SYSTEM DASDAass2_testi (* System Configuration *)
  (* Standard: 61499-1 *)
  (* Version 0.4, 2009-03-05, JHC, Holobloc Inc., Deleted Application. *)
  (* Version 0.3, 2003-12-05, JHC, Rockwell Automation, Renamed from NEWSYSTEM. *)
  (* Version 0.2, 2002-11-05, JHC, Rockwell Automation, Fixed missing (empty) FBD in Application. *)
  (* Version 0.1, 2002-01-17, JHC, Rockwell Automation, Minor cleanup *)
  (* Version 0.0, 2000-05-27, JHC, Rockwell Automation *)
  DEVICE HMI_LAYER : FRAME_DEVICE(BOUNDS := [0,0,200,200])
    RESOURCE HMI_1 : PANEL_RESOURCE(COLS := 1, ROWS := 0)
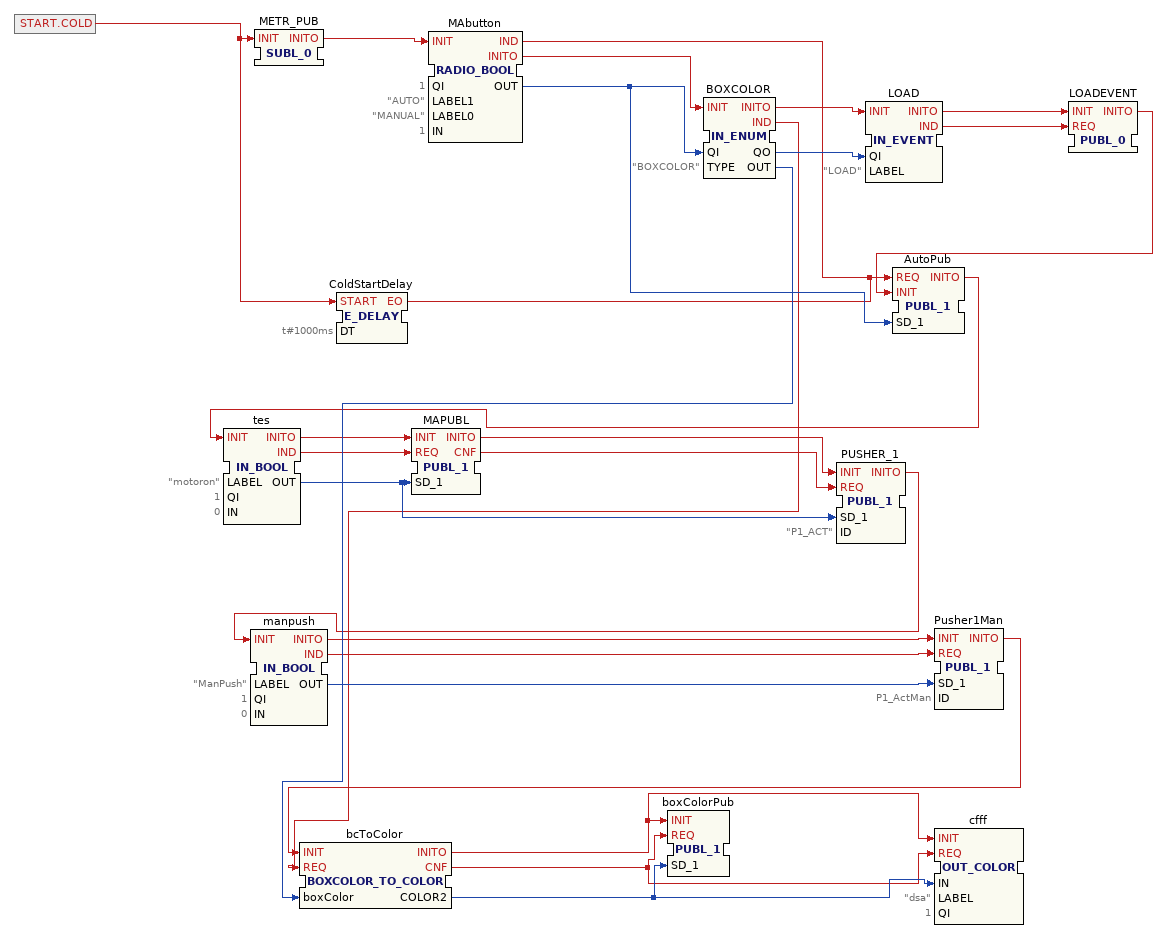
      FBS
        MAbutton : RADIO_BOOL(QI := 1, LABEL1 := "AUTO", LABEL0 := "MANUAL", IN := 1);
        LOAD : IN_EVENT(LABEL := "LOAD");
        LOADEVENT : PUBL_0;
        MAPUBL : PUBL_1;
        tes : IN_BOOL(LABEL := "motoron", QI := 1, IN := 0);
        METR_PUB : SUBL_0;
        PUSHER_1 : PUBL_1(ID := "P1_ACT");
        AutoPub : PUBL_1;
        ColdStartDelay : E_DELAY(DT := t#1000ms);
        manpush : IN_BOOL(LABEL := "ManPush", QI := 1, IN := 0);
        Pusher1Man : PUBL_1(ID := P1_ActMan);
        BOXCOLOR : IN_ENUM(TYPE := "BOXCOLOR");
        bcToColor : BOXCOLOR_TO_COLOR;
        cfff : OUT_COLOR(LABEL := "dsa", QI := 1);
        boxColorPub : PUBL_1;
      END_FBS
      EVENT_CONNECTIONS
        LOAD.INITO TO LOADEVENT.INIT;
        LOAD.IND TO LOADEVENT.REQ;
        START.COLD TO METR_PUB.INIT;
        METR_PUB.INITO TO MAbutton.INIT;
        tes.INITO TO MAPUBL.INIT;
        tes.IND TO MAPUBL.REQ;
        MAPUBL.INITO TO PUSHER_1.INIT;
        MAPUBL.CNF TO PUSHER_1.REQ;
        START.COLD TO ColdStartDelay.START;
        ColdStartDelay.EO TO AutoPub.REQ;
        MAbutton.IND TO AutoPub.REQ;
        LOADEVENT.INITO TO AutoPub.INIT;
        AutoPub.INITO TO tes.INIT;
        PUSHER_1.INITO TO manpush.INIT;
        manpush.INITO TO Pusher1Man.INIT;
        manpush.IND TO Pusher1Man.REQ;
        MAbutton.INITO TO BOXCOLOR.INIT;
        BOXCOLOR.INITO TO LOAD.INIT;
        Pusher1Man.INITO TO bcToColor.INIT;
        bcToColor.INITO TO cfff.INIT;
        bcToColor.CNF TO cfff.REQ;
        BOXCOLOR.IND TO bcToColor.REQ;
        bcToColor.INITO TO boxColorPub.INIT;
        bcToColor.CNF TO boxColorPub.REQ;
      END_CONNECTIONS
      DATA_CONNECTIONS
        tes.OUT TO MAPUBL.SD_1;
        tes.OUT TO PUSHER_1.SD_1;
        MAbutton.OUT TO AutoPub.SD_1;
        manpush.OUT TO Pusher1Man.SD_1;
        MAbutton.OUT TO BOXCOLOR.QI;
        BOXCOLOR.QO TO LOAD.QI;
        bcToColor.COLOR2 TO cfff.IN;
        BOXCOLOR.OUT TO bcToColor.boxColor;
        bcToColor.COLOR2 TO boxColorPub.SD_1;
      END_CONNECTIONS
    END_RESOURCE
  END_DEVICE
  DEVICE VIEW_LAYER : FRAME_DEVICE(BOUNDS := [250,0,900,900])
    RESOURCE VIEW_RES : VIEW_PANEL(DIA := 85, SIZE := [10,8], VERTICAL := 0)
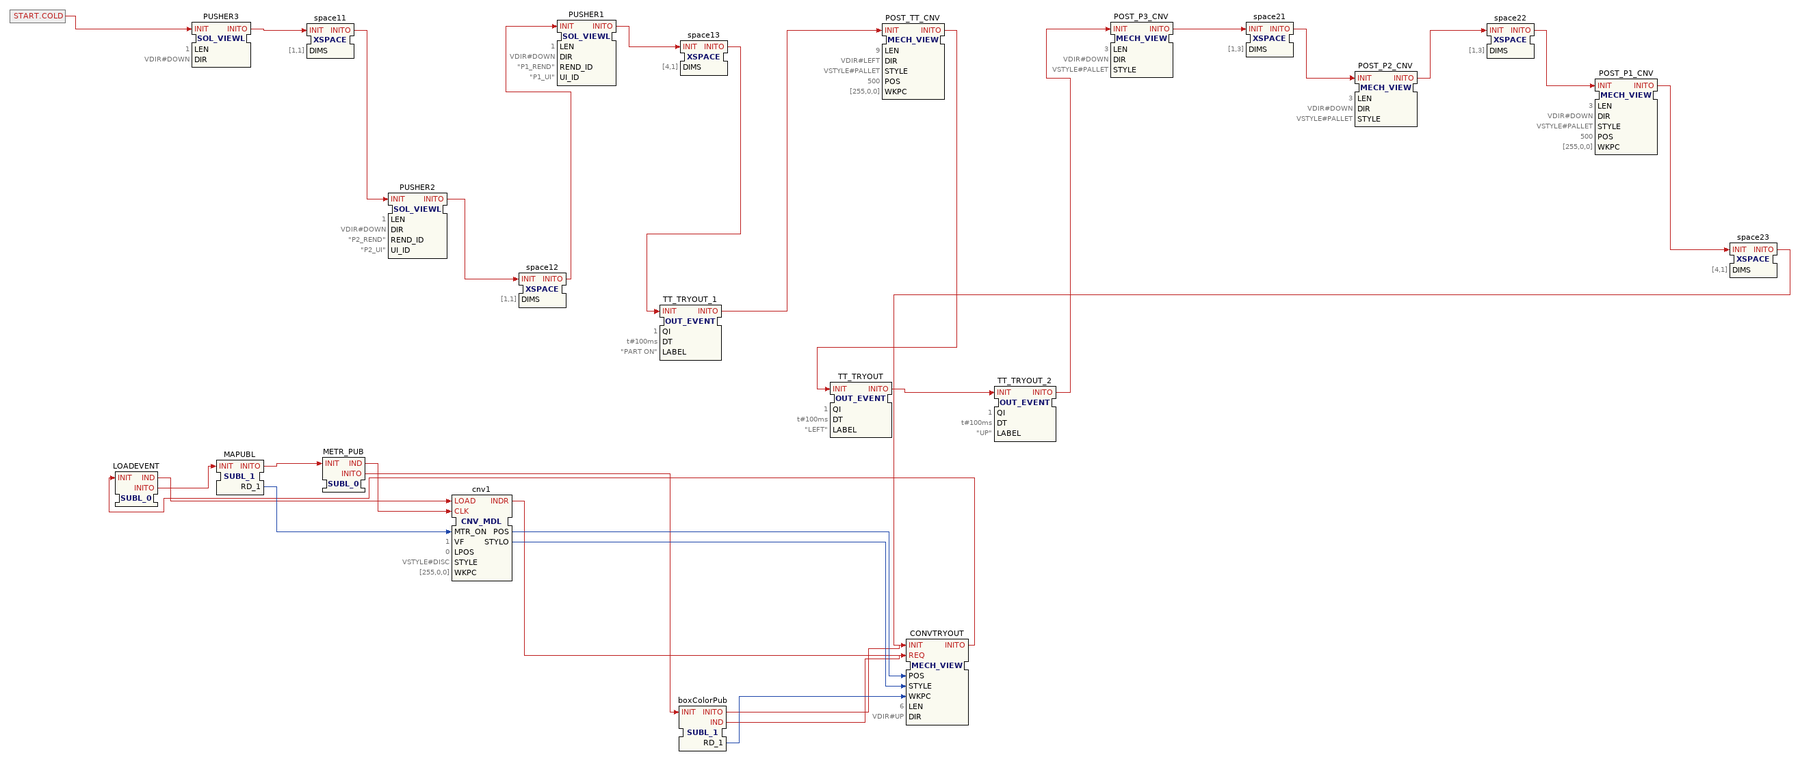
      FBS
        PUSHER3 : SOL_VIEWL(LEN := 1, DIR := VDIR#DOWN);
        space11 : XSPACE(DIMS := [1,1]);
        PUSHER2 : SOL_VIEWL(LEN := 1, DIR := VDIR#DOWN, REND_ID := "P2_REND", UI_ID := "P2_UI");
        space12 : XSPACE(DIMS := [1,1]);
        PUSHER1 : SOL_VIEWL(LEN := 1, DIR := VDIR#DOWN, REND_ID := "P1_REND", UI_ID := "P1_UI");
        space13 : XSPACE(DIMS := [4,1]);
        space21 : XSPACE(DIMS := [1,3]);
        space22 : XSPACE(DIMS := [1,3]);
        space23 : XSPACE(DIMS := [4,1]);
        POST_P1_CNV : MECH_VIEW(LEN := 3, DIR := VDIR#DOWN, STYLE := VSTYLE#PALLET, POS := 500, WKPC := [255,0,0]);
        POST_P2_CNV : MECH_VIEW(LEN := 3, DIR := VDIR#DOWN, STYLE := VSTYLE#PALLET);
        POST_P3_CNV : MECH_VIEW(LEN := 3, DIR := VDIR#DOWN, STYLE := VSTYLE#PALLET);
        POST_TT_CNV : MECH_VIEW(LEN := 9, DIR := VDIR#LEFT, STYLE := VSTYLE#PALLET, POS := 500, WKPC := [255,0,0]);
        TT_TRYOUT : OUT_EVENT(QI := 1, DT := t#100ms, LABEL := "LEFT");
        TT_TRYOUT_1 : OUT_EVENT(QI := 1, DT := t#100ms, LABEL := "PART ON");
        TT_TRYOUT_2 : OUT_EVENT(QI := 1, DT := t#100ms, LABEL := "UP");
        CONVTRYOUT : MECH_VIEW(LEN := 6, DIR := VDIR#UP);
        cnv1 : CNV_MDL(VF := 1, LPOS := 0, STYLE := VSTYLE#DISC, WKPC := [255,0,0]);
        LOADEVENT : SUBL_0;
        MAPUBL : SUBL_1;
        METR_PUB : SUBL_0;
        boxColorPub : SUBL_1;
      END_FBS
      EVENT_CONNECTIONS
        START.COLD TO PUSHER3.INIT;
        PUSHER3.INITO TO space11.INIT;
        space11.INITO TO PUSHER2.INIT;
        PUSHER2.INITO TO space12.INIT;
        space12.INITO TO PUSHER1.INIT;
        PUSHER1.INITO TO space13.INIT;
        space22.INITO TO POST_P1_CNV.INIT;
        POST_P1_CNV.INITO TO space23.INIT;
        space21.INITO TO POST_P2_CNV.INIT;
        POST_P2_CNV.INITO TO space22.INIT;
        POST_P3_CNV.INITO TO space21.INIT;
        POST_TT_CNV.INITO TO TT_TRYOUT.INIT;
        space13.INITO TO TT_TRYOUT_1.INIT;
        TT_TRYOUT_1.INITO TO POST_TT_CNV.INIT;
        TT_TRYOUT.INITO TO TT_TRYOUT_2.INIT;
        TT_TRYOUT_2.INITO TO POST_P3_CNV.INIT;
        space23.INITO TO CONVTRYOUT.INIT;
        CONVTRYOUT.INITO TO LOADEVENT.INIT;
        LOADEVENT.IND TO cnv1.LOAD;
        LOADEVENT.INITO TO MAPUBL.INIT;
        MAPUBL.INITO TO METR_PUB.INIT;
        METR_PUB.IND TO cnv1.CLK;
        cnv1.INDR TO CONVTRYOUT.REQ;
        boxColorPub.INITO TO CONVTRYOUT.INIT;
        boxColorPub.IND TO CONVTRYOUT.REQ;
        METR_PUB.INITO TO boxColorPub.INIT;
      END_CONNECTIONS
      DATA_CONNECTIONS
        cnv1.POS TO CONVTRYOUT.POS;
        cnv1.STYLO TO CONVTRYOUT.STYLE;
        MAPUBL.RD_1 TO cnv1.MTR_ON;
        boxColorPub.RD_1 TO CONVTRYOUT.WKPC;
      END_CONNECTIONS
    END_RESOURCE
  END_DEVICE
  DEVICE MODEL_LAYER : FRAME_DEVICE(BOUNDS := [0,200,200,200])
    RESOURCE MODEL_CLOCK : PANEL_RESOURCE
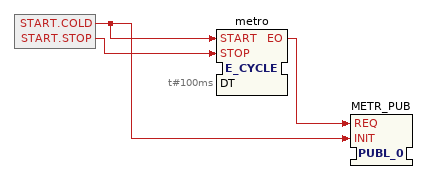
      FBS
        METR_PUB : PUBL_0;
        metro : E_CYCLE(DT := t#100ms);
      END_FBS
      EVENT_CONNECTIONS
        START.COLD TO metro.START;
        START.STOP TO metro.STOP;
        metro.EO TO METR_PUB.REQ;
        START.COLD TO METR_PUB.INIT;
      END_CONNECTIONS
    END_RESOURCE
    RESOURCE CNV_1_MODEL : PANEL_RESOURCE
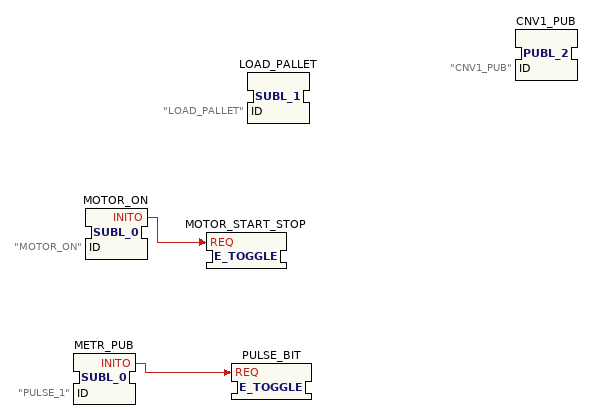
      FBS
        CNV1_PUB : PUBL_2(ID := "CNV1_PUB");
        METR_PUB : SUBL_0(ID := "PULSE_1");
        MOTOR_ON : SUBL_0(ID := "MOTOR_ON");
        LOAD_PALLET : SUBL_1(ID := "LOAD_PALLET");
        MOTOR_START_STOP : E_TOGGLE;
        PULSE_BIT : E_TOGGLE;
      END_FBS
      EVENT_CONNECTIONS
        MOTOR_ON.INITO TO MOTOR_START_STOP.REQ;
        METR_PUB.INITO TO PULSE_BIT.REQ;
      END_CONNECTIONS
    END_RESOURCE
    RESOURCE TT_MODEL : PANEL_RESOURCE
    END_RESOURCE
    RESOURCE CNV_2_MODEL : PANEL_RESOURCE
    END_RESOURCE
    RESOURCE PUSHER1_MODEL : PANEL_RESOURCE(ROWS := 0, COLS := 1)
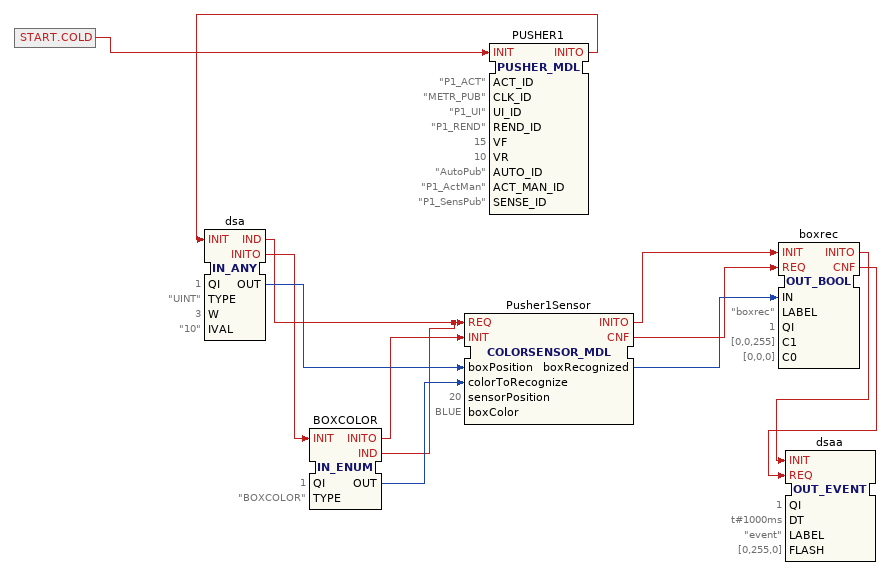
      FBS
        PUSHER1 : PUSHER_MDL(ACT_ID := "P1_ACT", CLK_ID := "METR_PUB", UI_ID := "P1_UI", REND_ID := "P1_REND", VF := 15, VR := 10, AUTO_ID := "AutoPub", ACT_MAN_ID := "P1_ActMan", SENSE_ID := "P1_SensPub");
        Pusher1Sensor : COLORSENSOR_MDL(sensorPosition := 20, boxColor := BLUE);
        dsa : IN_ANY(QI := 1, TYPE := "UINT", W := 3, IVAL := "10");
        boxrec : OUT_BOOL(LABEL := "boxrec", QI := 1, C1 := [0,0,255], C0 := [0,0,0]);
        dsaa : OUT_EVENT(QI := 1, DT := t#1000ms, LABEL := "event", FLASH := [0,255,0]);
        BOXCOLOR : IN_ENUM(QI := 1, TYPE := "BOXCOLOR");
      END_FBS
      EVENT_CONNECTIONS
        START.COLD TO PUSHER1.INIT;
        PUSHER1.INITO TO dsa.INIT;
        dsa.IND TO Pusher1Sensor.REQ;
        Pusher1Sensor.INITO TO boxrec.INIT;
        Pusher1Sensor.CNF TO boxrec.REQ;
        boxrec.INITO TO dsaa.INIT;
        boxrec.CNF TO dsaa.REQ;
        BOXCOLOR.INITO TO Pusher1Sensor.INIT;
        dsa.INITO TO BOXCOLOR.INIT;
        BOXCOLOR.IND TO Pusher1Sensor.REQ;
      END_CONNECTIONS
      DATA_CONNECTIONS
        dsa.OUT TO Pusher1Sensor.boxPosition;
        Pusher1Sensor.boxRecognized TO boxrec.IN;
        BOXCOLOR.OUT TO Pusher1Sensor.colorToRecognize;
      END_CONNECTIONS
    END_RESOURCE
    RESOURCE PUSHER_2_MODEL : PANEL_RESOURCE
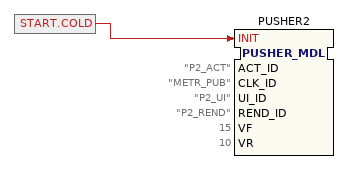
      FBS
        PUSHER2 : PUSHER_MDL(ACT_ID := "P2_ACT", CLK_ID := "METR_PUB", UI_ID := "P2_UI", REND_ID := "P2_REND", VF := 15, VR := 10);
      END_FBS
      EVENT_CONNECTIONS
        START.COLD TO PUSHER2.INIT;
      END_CONNECTIONS
    END_RESOURCE
    RESOURCE PUSHER3_MODEL : PANEL_RESOURCE
    END_RESOURCE
  END_DEVICE
END_SYSTEM
